SUBAPPLICATION mapping_TC_SC (* für TC-SC also Task Controller Section Control *)
  (* Standard: 61499-2 *)
  (* Version 1.0, 2023-10-23, franz *)
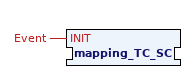
  EVENT_INPUT
    INIT;
  END_EVENT
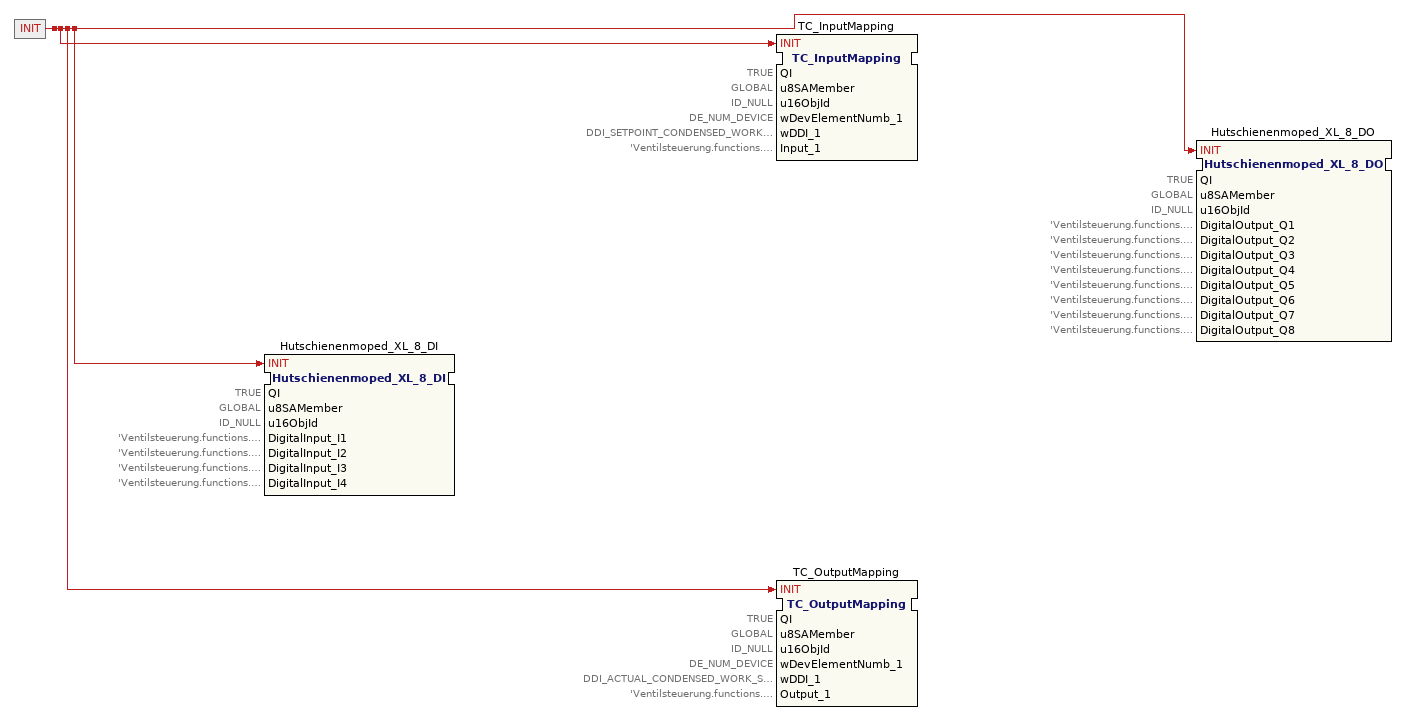
  FBS
    TC_InputMapping : TC_InputMapping(QI := TRUE, u8SAMember := GLOBAL, u16ObjId := ID_NULL, wDevElementNumb_1 := DE_NUM_DEVICE, wDDI_1 := DDI_SETPOINT_CONDENSED_WORK_STATE_1_16, Input_1 := 'Ventilsteuerung.functions.SETPOINT_CONDENSED_WORK_STATE_1_16');
    TC_OutputMapping : TC_OutputMapping(QI := TRUE, u8SAMember := GLOBAL, u16ObjId := ID_NULL, wDevElementNumb_1 := DE_NUM_DEVICE, wDDI_1 := DDI_ACTUAL_CONDENSED_WORK_STATE_1_16, Output_1 := 'Ventilsteuerung.functions.ACTUAL_CONDENSED_WORK_STATE_1_16');
    Hutschienenmoped_XL_8_DI : Hutschienenmoped_XL_8_DI(QI := TRUE, u8SAMember := GLOBAL, u16ObjId := ID_NULL, DigitalInput_I1 := 'Ventilsteuerung.functions.DigitalInput_I1', DigitalInput_I2 := 'Ventilsteuerung.functions.DigitalInput_I2', DigitalInput_I3 := 'Ventilsteuerung.functions.DigitalInput_I3', DigitalInput_I4 := 'Ventilsteuerung.functions.DigitalInput_I4');
    Hutschienenmoped_XL_8_DO : Hutschienenmoped_XL_8_DO(QI := TRUE, u8SAMember := GLOBAL, u16ObjId := ID_NULL, DigitalOutput_Q1 := 'Ventilsteuerung.functions.Out.DigitalOutput_Q1', DigitalOutput_Q2 := 'Ventilsteuerung.functions.Out.DigitalOutput_Q2', DigitalOutput_Q3 := 'Ventilsteuerung.functions.Out.DigitalOutput_Q3', DigitalOutput_Q4 := 'Ventilsteuerung.functions.Out.DigitalOutput_Q4', DigitalOutput_Q5 := 'Ventilsteuerung.functions.Out.DigitalOutput_Q5', DigitalOutput_Q6 := 'Ventilsteuerung.functions.Out.DigitalOutput_Q6', DigitalOutput_Q7 := 'Ventilsteuerung.functions.Out.DigitalOutput_Q7', DigitalOutput_Q8 := 'Ventilsteuerung.functions.Out.DigitalOutput_Q8');
  END_FBS
  EVENT_CONNECTIONS
    INIT TO TC_InputMapping.INIT;
    INIT TO TC_OutputMapping.INIT;
    INIT TO Hutschienenmoped_XL_8_DI.INIT;
    INIT TO Hutschienenmoped_XL_8_DO.INIT;
  END_CONNECTIONS
END_SUBAPPLICATION
